FUNCTION CheckVersion : BOOL
VAR_INPUT
	Major : UINT;
	Minor : UINT;
	Revision : UINT;
	Build : UINT;
END_VAR
VAR
END_VAR

IF Major = Version.Major
 AND Minor = Version.Minor
 AND Revision = Version.Revision
 AND Build = Version.Build
THEN
	CheckVersion := TRUE;
END_IF

END_FUNCTION

(* stored: Version 1.1.0.1, ProductVersion 3.1.4024.0
   POU CheckVersion: Id {9e2ddbef-7775-4a13-a318-40b2c35c443b}, SpecialFunc None *)
